(* Logix 5000 project; controller DUNEW2PLC1 vendor 1 type 14 code 221 rev 33.11; software revision 33.00; part 4 of 4 *)
(* tags used below, declared in another part *)
   INIT_DONE : BOOL;
   MOVE_TYPE : INT;   // 0 = No Move 1 = XY JOG 2 = XY Plane Move 3 = Z JOG 4 = Z Axis Move 5 = Toggle Latch Actuator 6 = Home the Latch Actuator
   NEXTSTATE : DINT;
   STATE : DINT;   // CURRENT State Machine State
   X_axis : AXIS_CIP_DRIVE;
   Y_axis : AXIS_CIP_DRIVE;
   Z_axis : AXIS_CIP_DRIVE;

PROGRAM UnServo_9   (* main routine UnServo_All *)
VAR
   oneshotob : BOOL[32]; {access Read Only}
   oneshotsb : BOOL[32]; {access Read Only}
   STATE9_IND : BOOL; {access Read Only}
   X_AXIS_STAT : MOTION_INSTRUCTION[32] := ([0].FLAGS := 33554432, [1].FLAGS := 33554432, [2].FLAGS := 536870912, [2].DN := 1, [2].STATE := 1); {access Read Only}
   Y_AXIS_STAT : MOTION_INSTRUCTION[32] := ([0].FLAGS := 33554432, [1].FLAGS := 33554432, [2].FLAGS := 536870912, [2].DN := 1, [2].STATE := 1); {access Read Only}
   Z_AXIS_STAT : MOTION_INSTRUCTION[32] := ([0].FLAGS := 33554432, [1].FLAGS := 33554432, [2].FLAGS := 536870912, [2].DN := 1, [2].STATE := 1); {access Read Only}
END_VAR

ROUTINE UnServo_All   (* ladder *)
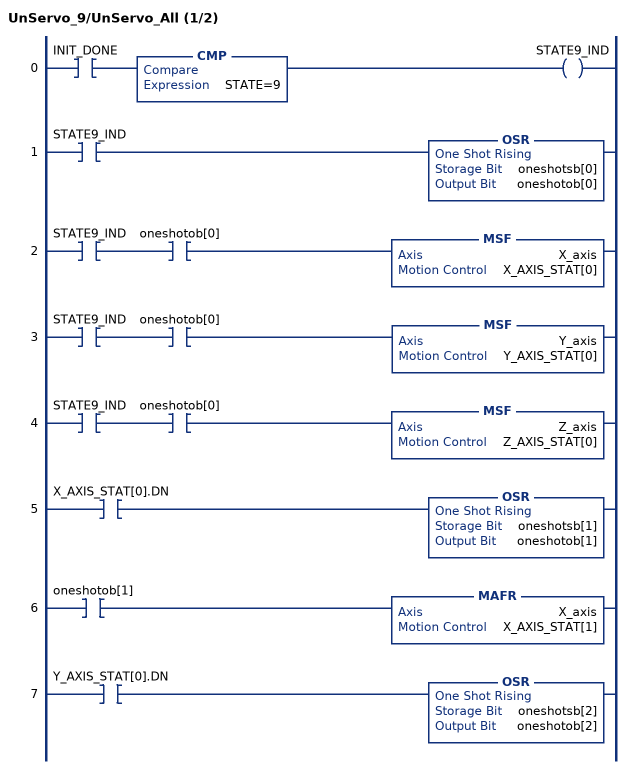
   0: XIC(INIT_DONE)CMP(STATE=9)OTE(STATE9_IND);
   1: XIC(STATE9_IND)OSR(oneshotsb[0],oneshotob[0]);
   2: XIC(STATE9_IND)XIC(oneshotob[0])MSF(X_axis,X_AXIS_STAT[0]);
   3: XIC(STATE9_IND)XIC(oneshotob[0])MSF(Y_axis,Y_AXIS_STAT[0]);
   4: XIC(STATE9_IND)XIC(oneshotob[0])MSF(Z_axis,Z_AXIS_STAT[0]);
   5: XIC(X_AXIS_STAT[0].DN)OSR(oneshotsb[1],oneshotob[1]);
   6: XIC(oneshotob[1])MAFR(X_axis,X_AXIS_STAT[1]);
   7: XIC(Y_AXIS_STAT[0].DN)OSR(oneshotsb[2],oneshotob[2]);
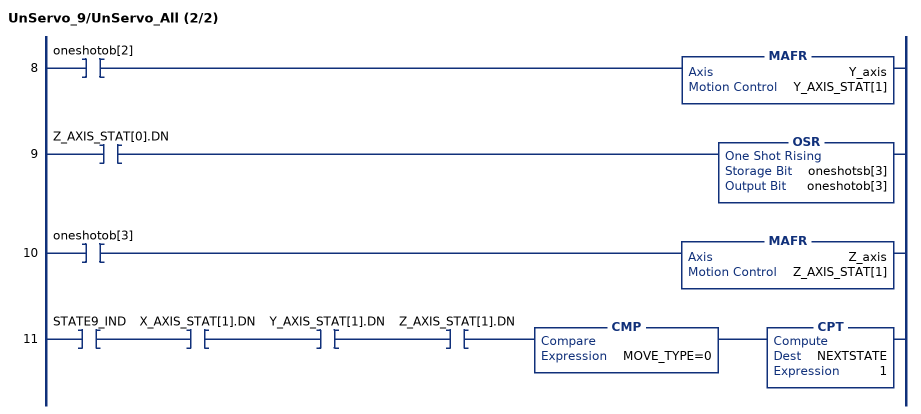
   8: XIC(oneshotob[2])MAFR(Y_axis,Y_AXIS_STAT[1]);
   9: XIC(Z_AXIS_STAT[0].DN)OSR(oneshotsb[3],oneshotob[3]);
   10: XIC(oneshotob[3])MAFR(Z_axis,Z_AXIS_STAT[1]);
   11: XIC(STATE9_IND)XIC(X_AXIS_STAT[1].DN)XIC(Y_AXIS_STAT[1].DN)XIC(Z_AXIS_STAT[1].DN)CMP(MOVE_TYPE=0)CPT(NEXTSTATE,1);
END_ROUTINE
END_PROGRAM
